(* CoDeSys 2.3 export: VARTYPE.EXP *)

(* Data type *)
TYPE VarType :
(
    BYTE_,
    WORD_,
    DWORD_,
    REAL_,
    DINT_,
    DWORD_30,
    DWORD_500
);
END_TYPE
